// TIA Portal V18 export
TYPE "PartDataHMI"
// stored: IsFailsafeCompliant false
   STRUCT
      PartQuality : DInt;   // 当前物料的剩余数量
      BoxDisplayID { S7_SetPoint := 'True'} : Int;   // 显示料盒编号
      PartQualitySet : DInt;   // 当前物料的剩余数量
      CMD : Struct   // 人工设定数量值
         ClearCurrentBox : Bool;
         ClearAllBox : Bool;
         "PartQuality+1" : Bool;
         "PartQuality-1" : Bool;
         PartQualityAck : Bool;   // 人工输入值确认
      END_STRUCT;
      Waring : Struct
         Insufficient : Bool;   // 物料不足，请扫码添加
         BufferBoxFull : Bool;   // 物料缓存已满，无法添加
         ScannCodeInvalid : Bool;   // 扫的物料码无效，或已经已用过
      END_STRUCT;
      PartDataDispaly : "PartCodeStruct_UDT";
   END_STRUCT;
END_TYPE
